PROGRAM z_LEVEL


(*-------------------------------------------------------------------------------------------------------*)
(*v038  Llenado nivel en caso de nivel por presion diferencial*)



(*-------------------------------------------------------------------------------------------------------*)
(*v039 valvula vaciado tubo nivel*)

END_PROGRAM

(* stored: Version 1.1.0.1, ProductVersion 3.1.4024.10
   POU z_LEVEL: Id {6a993ddb-2a84-478f-9096-bb4627b596db}, SpecialFunc None *)
